{attribute 'no_call'}
FUNCTION_BLOCK ABSTRACT FB_CyclicFB EXTENDS FB_BaseFB IMPLEMENTS I_CyclicFB
VAR
  _InitComplete : BOOL;
END_VAR

// Derivatives of FB_CyclicFB should *NOT* have code in the function block body

// Use CyclicLogic() instead

METHOD PUBLIC ABSTRACT CyclicLogic
VAR_INPUT
END_VAR
END_METHOD

PROPERTY InitComplete : BOOL
GET
InitComplete := _InitComplete;
END_GET
END_PROPERTY

END_FUNCTION_BLOCK

(* stored: Version 1.1.0.1, ProductVersion 3.1.4024.12
   POU FB_CyclicFB: Id {394075cc-3b9c-44ac-8717-5976ed11af50}, SpecialFunc None
   Folder I_CyclicFB: Id {15900726-6cfb-42d1-b875-3aa8d1a97c91}
   Method CyclicLogic: Id {6b9add30-ba72-4bcd-ae3f-b29cc64f5782}
   Property InitComplete: Id {ea567527-e93c-44d7-8358-003786bba1a3}
   Get Get: Id {c6fa949e-f03d-408b-8b5c-72f0d79338a7} *)
